(* IEC 61131-3 sources: CS_4_Aufzugsteuerung/src/Stations/CP112/Steuerung/Class/XXXBase_IOs, 1 file *)

(* ---- XXXBase_IOs.st ---- *)
(*!
<Class
	Name               = "XXXBase_IOs"
	Revision           = "1.2"
	RealtimeTask       = "false"
	CyclicTask         = "false"
	BackgroundTask     = "false"
	Sigmatek           = "true"
	OSInterface        = "false"
	HighPriority       = "false"
	Automatic          = "false"
	UpdateMode         = "Prescan"
	IconPath           = ".\Class\DigInOut.ICO"
	SharedCommandTable = "true"
	Objectsize         = "(570,540)"
	Comment            = "Baseclass for CPU_IO classes.">
	<Channels>
		<Server Name="CAN_1_Connect" Class="_CanLib" Visualized="false" Initialize="false" WriteProtected="true" Retentive="false" Comment="Connection servers for Hardware-Editor."/>
		<Server Name="CAN_2_Connect" Class="_CanLib" Visualized="false" Initialize="false" WriteProtected="true" Retentive="false" Comment="Connection servers for Hardware-Editor."/>
		<Server Name="ClassState" Visualized="true" Initialize="false" WriteProtected="true" Retentive="false" Comment="Shows the state of the class.&#13;&#10;0 ... ok."/>
		<Server Name="COM_1_Connect" Class="_SerLib" Visualized="false" Initialize="false" WriteProtected="true" Retentive="false" Comment="Connection servers for Hardware-Editor."/>
		<Server Name="COM_2_Connect" Class="_SerLib" Visualized="false" Initialize="false" WriteProtected="true" Retentive="false" Comment="Connection servers for Hardware-Editor."/>
		<Server Name="COM_3_Connect" Class="_SerLib" Visualized="false" Initialize="false" WriteProtected="true" Retentive="false" Comment="Connection servers for Hardware-Editor."/>
		<Server Name="Ethernet_1_Connect" Visualized="false" Initialize="false" WriteProtected="true" Retentive="false" Comment="Connection servers for Hardware-Editor."/>
		<Server Name="Ethernet_2_Connect" Visualized="false" Initialize="false" WriteProtected="true" Retentive="false" Comment="Connection servers for Hardware-Editor."/>
		<Server Name="Ethernet_3_Connect" Visualized="false" Initialize="false" WriteProtected="true" Retentive="false" Comment="Connection servers for Hardware-Editor."/>
		<Server Name="Ethernet_4_Connect" Visualized="false" Initialize="false" WriteProtected="true" Retentive="false" Comment="Connection servers for Hardware-Editor."/>
		<Server Name="USB_1_Connect" Visualized="false" Initialize="false" WriteProtected="true" Retentive="false" Comment="Connection servers for Hardware-Editor."/>
		<Client Name="_CanLib1" Required="true" Internal="true"/>
		<Client Name="_CanLib2" Required="true" Internal="true"/>
		<Client Name="_SerLib1" Required="true" Internal="true"/>
		<Client Name="_SerLib2" Required="true" Internal="true"/>
		<Client Name="_SerLib3" Required="true" Internal="true"/>
		<Client Name="To_HwControl" Required="true" Internal="false" Comment="Connect to server &quot;Control&quot; of &quot;HwControl&quot;-Object"/>
	</Channels>
	<RevDoku>
		<Owner Company="Sigmatek" Author="HaeTho"/>
		<Dokumentation Revision="1.2" Date="2025-11-03" Author="ZoeJoh" Company="Sigmatek" Description="Method LogValue last 2 parameter initialized"/>
		<Dokumentation Revision="1.1" Date="06.11.2018" Author="HaeTho&#13;&#10;EisMic" Company="Sigmatek" Description="Index of sub classes for CAN- and seriell connection is now &gt;= 1&#13;&#10;Added methods LogError and LogValue."/>
		<Dokumentation Revision="1.0" Date="02.08.2018" Author="HaeTho" Company="Sigmatek" Description="Hardware-Editor Bus-Connectors, first library version"/>
	</RevDoku>
	<Network Name="XXXBase_IOs">
		<!-- List of Components in this network -->
		<Components>
			<Object
				Name       = "_CanLib1"
				Class      = "_CanLib"
				Position   = "(150,300)"
				Visualized = "true"
				Remotely   = "true">
				<Channels>
					<Server Name="CanBus" Value="1"/>
					<Server Name="Command"/>
					<Client Name="To_Can"/>
				</Channels>
			</Object>
			<Object
				Name       = "_CanLib2"
				Class      = "_CanLib"
				Position   = "(150,510)"
				Visualized = "true"
				Remotely   = "true">
				<Channels>
					<Server Name="CanBus" Value="2"/>
					<Server Name="Command"/>
					<Client Name="To_Can"/>
				</Channels>
			</Object>
			<Object
				Name       = "_SerLib1"
				Class      = "_SerLib"
				Position   = "(150,720)"
				Visualized = "true"
				Remotely   = "true">
				<Channels>
					<Server Name="Com" Value="1"/>
					<Server Name="Command"/>
				</Channels>
			</Object>
			<Object
				Name       = "_SerLib2"
				Class      = "_SerLib"
				Position   = "(150,930)"
				Visualized = "true"
				Remotely   = "true">
				<Channels>
					<Server Name="Com" Value="2"/>
					<Server Name="Command"/>
				</Channels>
			</Object>
			<Object
				Name       = "_SerLib3"
				Class      = "_SerLib"
				Position   = "(150,1140)"
				Visualized = "true"
				Remotely   = "true">
				<Channels>
					<Server Name="Com" Value="3"/>
					<Server Name="Command"/>
				</Channels>
			</Object>
		</Components>
		<Comments>
		</Comments>
		<!-- List of Connections in this network -->
		<Connections>
			<Connection Source="this._CanLib1" Destination="_CanLib1.Command"/>
			<Connection Source="this.CAN_1_Connect" Destination="_CanLib1.Command" Vertices="(652,570),(480,390),"/>
			<Connection Source="this._CanLib2" Destination="_CanLib2.Command"/>
			<Connection Source="this.CAN_2_Connect" Destination="_CanLib2.Command" Vertices="(652,630),(480,600),"/>
			<Connection Source="this._SerLib1" Destination="_SerLib1.Command"/>
			<Connection Source="this.COM_1_Connect" Destination="_SerLib1.Command" Vertices="(652,690),(450,810),"/>
			<Connection Source="this._SerLib2" Destination="_SerLib2.Command"/>
			<Connection Source="this.COM_2_Connect" Destination="_SerLib2.Command" Vertices="(652,750),(450,1020),"/>
			<Connection Source="this._SerLib3" Destination="_SerLib3.Command"/>
			<Connection Source="this.COM_3_Connect" Destination="_SerLib3.Command" Vertices="(652,810),(450,1230),"/>
		</Connections>
		<!-- Headerfiles -->
		<Options>
		</Options>
	</Network>
</Class>
*)
XXXBase_IOs : CLASS
  //Servers:
	ClassState 	: SvrChCmd_DINT;
	USB_1_Connect 	: SvrChCmd_DINT;
	Ethernet_1_Connect 	: SvrChCmd_DINT;
	Ethernet_2_Connect 	: SvrChCmd_DINT;
	Ethernet_3_Connect 	: SvrChCmd_DINT;
	Ethernet_4_Connect 	: SvrChCmd_DINT;
	CAN_1_Connect 	: SvrChCmd_DINT;
	CAN_2_Connect 	: SvrChCmd_DINT;
	COM_1_Connect 	: SvrChCmd_DINT;
	COM_2_Connect 	: SvrChCmd_DINT;
	COM_3_Connect 	: SvrChCmd_DINT;
  //Clients:
	To_HwControl 	: CltChCmd_HwControl;
	_SerLib1 	: CltChCmd__SerLib;
	_SerLib2 	: CltChCmd__SerLib;
	_CanLib1 	: CltChCmd__CanLib;
	_CanLib2 	: CltChCmd__CanLib;
	_SerLib3 	: CltChCmd__SerLib;
  //Variables:
  //Functions:

	FUNCTION LogError
		VAR_INPUT
			pMsg 	: ^CHAR;
		END_VAR;

	FUNCTION LogValue
		VAR_INPUT
			pString 	: ^CHAR;
			udValue 	: UDINT;
			udValue2 	: UDINT := 16#FFFFFFFF;
			udValue3 	: UDINT := 16#FFFFFFFF;
		END_VAR;

	FUNCTION VIRTUAL GLOBAL Ethernet_1_Connect::NewInst
		VAR_INPUT
			pPara 	: ^CmdStruct;
			pResult 	: ^results;
		END_VAR
		VAR_OUTPUT
			ret_code 	: iprStates;
		END_VAR;

	FUNCTION VIRTUAL GLOBAL Ethernet_2_Connect::NewInst
		VAR_INPUT
			pPara 	: ^CmdStruct;
			pResult 	: ^results;
		END_VAR
		VAR_OUTPUT
			ret_code 	: iprStates;
		END_VAR;

	FUNCTION VIRTUAL GLOBAL Ethernet_3_Connect::NewInst
		VAR_INPUT
			pPara 	: ^CmdStruct;
			pResult 	: ^results;
		END_VAR
		VAR_OUTPUT
			ret_code 	: iprStates;
		END_VAR;

	FUNCTION VIRTUAL GLOBAL Ethernet_4_Connect::NewInst
		VAR_INPUT
			pPara 	: ^CmdStruct;
			pResult 	: ^results;
		END_VAR
		VAR_OUTPUT
			ret_code 	: iprStates;
		END_VAR;

	FUNCTION VIRTUAL GLOBAL COM_3_Connect::Read
		VAR_OUTPUT
			output (EAX) 	: DINT;
		END_VAR;
  //Tables:
	FUNCTION @STD
		VAR_OUTPUT
			ret_code	: CONFSTATES;
		END_VAR;
	FUNCTION GLOBAL TAB @CT_;
END_CLASS;

#pragma using _CanLib
#pragma using _SerLib
#pragma usingLtd HwControl

FUNCTION XXXBase_IOs::LogError
	VAR_INPUT
		pMsg 	: ^CHAR;
	END_VAR

#ifdef HWC_LogError
  HWC_LogError(this, pMsg);
#endif

END_FUNCTION

FUNCTION XXXBase_IOs::LogValue
	VAR_INPUT
		pString 	: ^CHAR;
		udValue 	: UDINT;
		udValue2 	: UDINT;(* := 16#FFFFFFFF *)
		udValue3 	: UDINT;(* := 16#FFFFFFFF *)
	END_VAR

#ifdef HWC_LogValue3
  HWC_LogValue3(this, pString, udValue, udValue2, udValue3);
#endif

END_FUNCTION

FUNCTION VIRTUAL GLOBAL XXXBase_IOs::Ethernet_1_Connect::NewInst
	VAR_INPUT
		pPara 	: ^CmdStruct;
		pResult 	: ^Results;
	END_VAR
	VAR_OUTPUT
		ret_code 	: IprStates;
	END_VAR

  ret_code := ERROR;

	CASE pPara^.uiCmd OF

    //***********************************************************************************************************
		CMD_HWC_GET_INTERFACE_NUMBER:

      //Check for valid version
      if pPara^.aPara[0] = 0x1 then

        //Return version number
        pResult^.aData[0] := 0x1;

        //Interface number of Ethernet Interface
        pResult^.aData[1]$DINT  := 1;

        ret_code := READY;
      end_if;

    //***********************************************************************************************************

	END_CASE;

END_FUNCTION

FUNCTION VIRTUAL GLOBAL XXXBase_IOs::Ethernet_2_Connect::NewInst
	VAR_INPUT
		pPara 	: ^CmdStruct;
		pResult 	: ^Results;
	END_VAR
	VAR_OUTPUT
		ret_code 	: IprStates;
	END_VAR

  ret_code := ERROR;

	CASE pPara^.uiCmd OF

    //***********************************************************************************************************
		CMD_HWC_GET_INTERFACE_NUMBER:

      //Check for valid version
      if pPara^.aPara[0] = 0x1 then

        //Return version number
        pResult^.aData[0] := 0x1;

        //Interface number of Ethernet Interface
        pResult^.aData[1]$DINT  := 2;

        ret_code := READY;
      end_if;

    //***********************************************************************************************************

	END_CASE;

END_FUNCTION

FUNCTION VIRTUAL GLOBAL XXXBase_IOs::Ethernet_3_Connect::NewInst
	VAR_INPUT
		pPara 	: ^CmdStruct;
		pResult 	: ^Results;
	END_VAR
	VAR_OUTPUT
		ret_code 	: IprStates;
	END_VAR

  ret_code := ERROR;

	CASE pPara^.uiCmd OF

    //***********************************************************************************************************
		CMD_HWC_GET_INTERFACE_NUMBER:

      //Check for valid version
      if pPara^.aPara[0] = 0x1 then

        //Return version number
        pResult^.aData[0] := 0x1;

        //Interface number of Ethernet Interface
        pResult^.aData[1]$DINT  := 3;

        ret_code := READY;
      end_if;

    //***********************************************************************************************************

	END_CASE;

END_FUNCTION

FUNCTION VIRTUAL GLOBAL XXXBase_IOs::Ethernet_4_Connect::NewInst
	VAR_INPUT
		pPara 	: ^CmdStruct;
		pResult 	: ^Results;
	END_VAR
	VAR_OUTPUT
		ret_code 	: IprStates;
	END_VAR

  ret_code := ERROR;

	CASE pPara^.uiCmd OF

    //***********************************************************************************************************
		CMD_HWC_GET_INTERFACE_NUMBER:

      //Check for valid version
      if pPara^.aPara[0] = 0x1 then

        //Return version number
        pResult^.aData[0] := 0x1;

        //Interface number of Ethernet Interface
        pResult^.aData[1]$DINT  := 4;

        ret_code := READY;
      end_if;

    //***********************************************************************************************************

	END_CASE;

END_FUNCTION

FUNCTION VIRTUAL GLOBAL XXXBase_IOs::COM_3_Connect::Read
	VAR_OUTPUT
		output (EAX) 	: DINT;
	END_VAR

	COM_3_Connect := _SerLib3.Command.Read();
	output := COM_3_Connect;

END_FUNCTION
